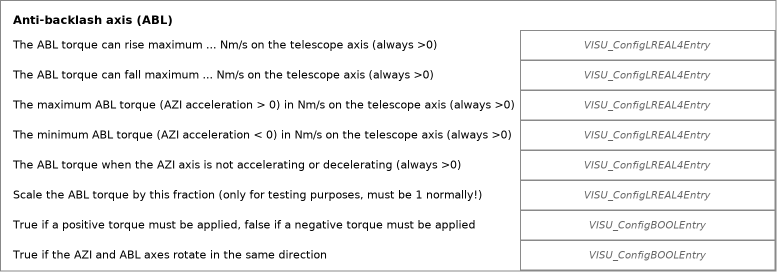
VISUALIZATION VISU_AxesConfig_Azimuth_3  // 777x272
VAR_IN_OUT
    active : AxesAzimuthConfig;
    editable : AxesAzimuthConfig;
END_VAR
    Label (10,5 205x30), "Anti-backlash axis (ABL)"
    Label (10,30 475x30), "The ABL torque can rise maximum ... Nm/s on the telescope axis (always >0)"
    Frame (520,30 255x30)
        shows VISU_ConfigLREAL4Entry(active := active.ablMaxTorqueRiseSpeed, editable := editable.ablMaxTorqueRiseSpeed)
    Label (10,60 475x30), "The ABL torque can fall maximum ... Nm/s on the telescope axis (always >0)"
    Label (10,90 505x30), "The maximum ABL torque (AZI acceleration > 0) in Nm/s on the telescope axis (always >0)"
    Label (10,120 500x30), "The minimum ABL torque (AZI acceleration < 0) in Nm/s on the telescope axis (always >0)"
    Label (10,150 500x30), "The ABL torque when the AZI axis is not accelerating or decelerating (always >0)"
    Label (10,180 500x30), "Scale the ABL torque by this fraction (only for testing purposes, must be 1 normally!)"
    Label (10,210 500x30), "True if a positive torque must be applied, false if a negative torque must be applied"
    Frame (520,210 255x30)
        shows VISU_ConfigBOOLEntry(active := active.ablPositiveTorque, editable := editable.ablPositiveTorque)
    Label (10,240 500x30), "True if the AZI and ABL axes rotate in the same direction"
    Frame (520,240 255x30)
        shows VISU_ConfigBOOLEntry(active := active.aziAndAblSameDirection, editable := editable.aziAndAblSameDirection)
    Frame (520,60 255x30)
        shows VISU_ConfigLREAL4Entry(active := active.ablMaxTorqueFallSpeed, editable := editable.ablMaxTorqueFallSpeed)
    Frame (520,90 255x30)
        shows VISU_ConfigLREAL4Entry(active := active.ablMaxTorque, editable := editable.ablMaxTorque)
    Frame (520,120 255x30)
        shows VISU_ConfigLREAL4Entry(active := active.ablMinTorque, editable := editable.ablMinTorque)
    Frame (520,150 255x30)
        shows VISU_ConfigLREAL4Entry(active := active.ablZeroAccTorque, editable := editable.ablZeroAccTorque)
    Frame (520,180 255x30)
        shows VISU_ConfigLREAL4Entry(active := active.ablTorqueOutputOverride, editable := editable.ablTorqueOutputOverride)
END_VISUALIZATION

(* stored: Version 1.1.0.1, ProductVersion 3.1.4019.2
   Visu VISU_AxesConfig_Azimuth_3: Id {67b141c7-e13f-413e-9e05-91e44981c21e} *)
